FUNCTION_BLOCK PusherControl (* Basic Function Block Type *)
  (* Standard: 61499-2 *)
  (* Version 0.0, 1/14/2024, midxav, Template *)
  PACKAGE Main;
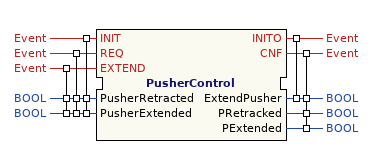
  EVENT_INPUT
    INIT WITH PusherRetracted, PusherExtended; (* Initialization Request *)
    REQ WITH PusherRetracted, PusherExtended; (* Normal Execution Request *)
    EXTEND WITH PusherRetracted, PusherExtended;
  END_EVENT
  EVENT_OUTPUT
    INITO WITH ExtendPusher; (* Initialization Confirm *)
    CNF WITH ExtendPusher, PRetracked, PExtended; (* Execution Confirmation *)
  END_EVENT
  VAR_INPUT
    PusherRetracted : BOOL;
    PusherExtended : BOOL;
  END_VAR
  VAR_OUTPUT
    ExtendPusher : BOOL;
    PRetracked : BOOL;
    PExtended : BOOL;
  END_VAR
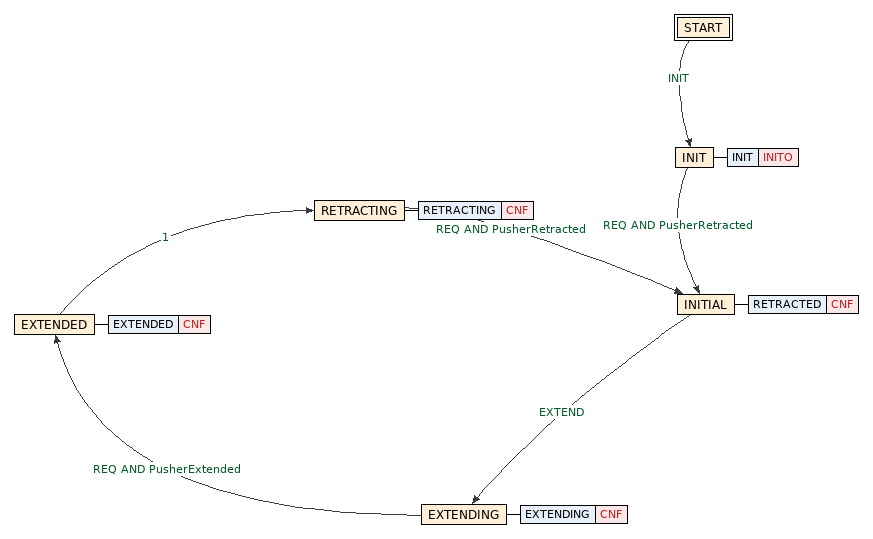
  EC_STATES
    START; (* Initial State *)
    INIT : INIT -> INITO; (* Initialization *)
    INITIAL : RETRACTED -> CNF;
    EXTENDING : EXTENDING -> CNF;
    EXTENDED : EXTENDED -> CNF;
    RETRACTING : RETRACTING -> CNF;
  END_STATES
  EC_TRANSITIONS
    START TO INIT := INIT;
    INIT TO INITIAL := REQ AND PusherRetracted;
    EXTENDING TO EXTENDED := REQ AND PusherExtended;
    INITIAL TO EXTENDING := EXTEND;
    EXTENDED TO RETRACTING := 1;
    RETRACTING TO INITIAL := REQ AND PusherRetracted;
  END_TRANSITIONS
  ALGORITHM INIT IN ST: (* Initialization algorithm *)
ExtendPusher:= FALSE;
PRetracked:= FALSE;
PExtended := FALSE;
  END_ALGORITHM
  ALGORITHM EXTENDING IN ST:
ExtendPusher:=TRUE;
PRetracked:=FALSE;
  END_ALGORITHM
  ALGORITHM EXTENDED IN ST:
ExtendPusher:=FALSE;
PExtended:=TRUE;
  END_ALGORITHM
  ALGORITHM RETRACTED IN ST:
;
PRetracked:= TRUE;
  END_ALGORITHM
  ALGORITHM RETRACTING IN ST:
PExtended:= FALSE;
  END_ALGORITHM
END_FUNCTION_BLOCK
